# EPICS autosave request: tests/testfiles/cfg/SF_timing_PulDel_PV.req
$(SYS)-EVR0:Pul0-Delay-SP
$(SYS)-EVR0:Pul1-Delay-SP
$(SYS)-EVR0:Pul2-Delay-SP
$(SYS)-EVR0:Pul3-Delay-SP
$(SYS)-EVR0:Pul4-Delay-SP
$(SYS)-EVR0:Pul5-Delay-SP
$(SYS)-EVR0:Pul6-Delay-SP
$(SYS)-EVR0:Pul7-Delay-SP
$(SYS)-EVR0:Pul8-Delay-SP
$(SYS)-EVR0:Pul9-Delay-SP
$(SYS)-EVR0:Pul10-Delay-SP
$(SYS)-EVR0:Pul11-Delay-SP
$(SYS)-EVR0:Pul12-Delay-SP
$(SYS)-EVR0:Pul13-Delay-SP
$(SYS)-EVR0:Pul14-Delay-SP
$(SYS)-EVR0:Pul15-Delay-SP
$(SYS)-EVR0:Pul16-Delay-SP
$(SYS)-EVR0:Pul17-Delay-SP
$(SYS)-EVR0:Pul18-Delay-SP
$(SYS)-EVR0:Pul19-Delay-SP
$(SYS)-EVR0:Pul20-Delay-SP
$(SYS)-EVR0:Pul21-Delay-SP
$(SYS)-EVR0:Pul22-Delay-SP
$(SYS)-EVR0:Pul23-Delay-SP
